(* IEC 61131-3 sources: codefinetuner/third_party/tree-sitter-iec61131-3-st/examples/dialect-extension, 1 file *)

(* ---- sample.st ---- *)
(*
 * Sample TwinCAT-flavored ST that exercises the dialect's extensions.
 *)

PROGRAM SystemReader
VAR
    task_idx : DINT;
    safe     : BOOL;
    p        : POINTER TO INT;
    val      : INT;
END_VAR

task_idx := __SYSTEM.GetCurrentTaskIndex();

(* Short-circuit AND_THEN: only dereference p if it's non-NULL. *)
safe := (p <> 0) AND_THEN (p^ > 0);
IF safe THEN
    val := p^;
END_IF
END_PROGRAM
